// TIA Portal project "Project2" (V16)

(* hardware
DEVICE "S7-1200 station_1"  S7-1200 Station
   slot 0: "Rack_0"  S7-1200 Rack  Rack  V1.0
   slot 1: "PLC_1"  CPU 1212C AC/DC/Rly  6ES7 212-1BE40-0XB0  V4.4
*)

// ===== PLC "PLC_1"  CPU 1212C AC/DC/Rly =====

ORGANIZATION_BLOCK "Main"   // OB1, LAD, ProgramCycle
TITLE = "Main Program Sweep (Cycle)"
{ S7_Optimized_Access := 'TRUE' }
VERSION : 0.1
   VAR_INPUT
      Initial_Call : Bool;   // Initial call of this OB
      Remanence : Bool;   // =True, if remanent data are available
   END_VAR
BEGIN

REGION Network 1
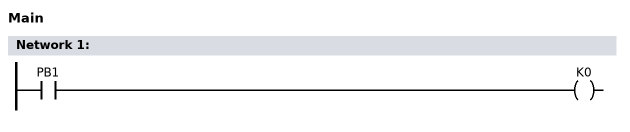
   RUNG wire#powerrail
      Contact( PB1 )
      Coil( K0 )
   END_RUNG
   RUNG wire#powerrail
   END_RUNG
   // the same network as SCL:
   K0 := PB1;
END_REGION
END_ORGANIZATION_BLOCK